TYPE
    ST_AllocateStatus :
    STRUCT
    END_STRUCT
END_TYPE

(* stored: Version 1.1.0.1, ProductVersion 3.1.4024.13
   DUT ST_AllocateStatus: Id {0a8bf2e5-b109-4ac9-87df-66582705487c} *)
